FUNCTION_BLOCK MyCalculatorClass
VAR
END_VAR

METHOD Divide : INT
VAR_INPUT
	x : INT;
	y : INT;
END_VAR
IF y <> 0 THEN
	Divide := x/y;
ELSE
	Divide := -1;
END_IF
END_METHOD

END_FUNCTION_BLOCK

(* stored: Version 1.1.0.1, ProductVersion 3.1.4024.12
   POU MyCalculatorClass: Id {d0dae815-f97c-4665-8a1f-5832f41e610e}, SpecialFunc None
   Method Divide: Id {a41cb6fc-1473-45fd-9cff-c951ededf815} *)
